TYPE ST_ServiceRegistrationEntry :
STRUCT
	InUse : BOOL;
	ServiceId : UDINT;

	UpperCtrlAddress : PVOID;
	EffectiveCtrlAddress : PVOID;

	UpperParamAddress : PVOID;
	EffectiveParamAddress : PVOID;
	ParameterSize : UDINT;
	ParameterTypeName : STRING(255);

	StatusAddress : PVOID;

	UpperCommandWasHigh : BOOL;
	UpperModeWasHigh : BOOL;
	UpperCommandBlockedUntilFalse : BOOL;
	UpperModeBlockedUntilFalse : BOOL;
END_STRUCT
END_TYPE

(* stored: Version 1.1.0.1, ProductVersion 3.1.4026.18
   DUT ST_ServiceRegistrationEntry: Id {77e6d734-5908-45a5-ad5f-d5db1cdf75b0} *)
